{attribute 'qualified_only'}
VAR_GLOBAL

	sDevice					: ST_IoT_Device_General;
	sRooms					: ST_IoT_HMI_Rooms;

END_VAR

(* stored: Version 1.1.0.1, ProductVersion 3.1.4024.12
   GVL GVL_HMI: Id {ce3e895e-8be5-497e-a143-3ff8049dec87} *)
